// Example of "device-to-device" communication.
// [Notes]
// > Apply devices routes via "Diangnose / Device communication" in TerminalExplorer when PLC's are in run-mode.
//   Afterwards all communication errors will disappear. 
FUNCTION_BLOCK FB_Ref_PubSub_Remote EXTENDS FB_BA_View
VAR CONSTANT
	{region 'Test Settings'}
		// Use one (remote) device:
//		sDevice1_NetID			: T_BA_MedString				:= '192.168.10.100.1.1';
//		sDevice2_NetID			: T_BA_MedString				:= '192.168.10.100.1.1';
			 
		// Use one (loopback) device:
		sDevice1_NetID			: T_BA_MedString				:= '127.0.0.1.1.1';
		sDevice2_NetID			: T_BA_MedString				:= '127.0.0.1.1.1';
			 
		// Use two (remote and loopback) devices:
//		sDevice1_NetID			: T_BA_MedString				:= '192.168.2.200.1.1';
//		sDevice2_NetID			: T_BA_MedString				:= '127.0.0.1.1.1';
			 
		// Use two (remote) devices:
//		sDevice1_NetID			: T_BA_MedString				:= '192.168.10.100.1.1';
//		sDevice2_NetID			: T_BA_MedString				:= '192.168.2.200.1.1';
	{endregion}
END_VAR
VAR
	{region 'Analog'}
		AV_Sub					: FB_BA_SubAPrio := (
									sSubject					:= 'AV_Obj',
									sTarget						:= sDevice1_NetID,
									tReadInterval				:= T#5S								// Set shorter read interval
								);
		AVOp_Sub				: FB_BA_SubAV_Op := (
									sSubject					:= 'AVOp_Obj',
									sTarget						:= sDevice1_NetID,
									tReadInterval				:= T#5S								// Set shorter read interval
								);
		AI_Sub					: FB_BA_SubAI := (
									sSubject					:= 'AI_Obj',
									sTarget						:= sDevice2_NetID,
									tReadInterval				:= T#5S								// Set shorter read interval
								);
		AO_Sub					: FB_BA_SubAPrio := (
									sSubject					:= 'AO_Obj',
									sTarget						:= sDevice2_NetID,
									tReadInterval				:= T#5S								// Set shorter read interval
								);
	{endregion}
	{region 'Binary'}
		BV_Sub					: FB_BA_SubBPrio := (
									sSubject					:= 'BV_Obj',
									sTarget						:= sDevice1_NetID
								);
		BVOp_Sub				: FB_BA_SubBV_Op := (
									sSubject					:= 'BVOp_Obj',
									sTarget						:= sDevice1_NetID
								);
		BI_Sub					: FB_BA_SubBI := (
									sSubject					:= 'BI_Obj',
									sTarget						:= sDevice2_NetID
								);
		BO_Sub					: FB_BA_SubBPrio := (
									sSubject					:= 'BO_Obj',
									sTarget						:= sDevice2_NetID
								);
	{endregion}
	{region 'Multistate'}
		MV_Sub					: FB_BA_SubMPrio := (
									sSubject					:= 'MV_Obj',
									sTarget						:= sDevice1_NetID
								);
		MVOp_Sub				: FB_BA_SubMV_Op := (
									sSubject					:= 'MVOp_Obj',
									sTarget						:= sDevice1_NetID
								);
		MI_Sub					: FB_BA_SubMI := (
									sSubject					:= 'MI_Obj',
									sTarget						:= sDevice2_NetID
								);
		MO_Sub					: FB_BA_SubMPrio := (
									sSubject					:= 'MO_Obj',
									sTarget						:= sDevice2_NetID
								);
	{endregion}
	{region 'Multistate'}
		Loop_Sub				: FB_BA_SubLoop := (
									sSubject					:= 'Loop_Obj',
									sTarget						:= sDevice1_NetID
								);		
		Cal_Sub					: FB_BA_SubCal := (
									sSubject					:= 'Cal_Obj',
									sTarget						:= sDevice1_NetID
								);
		SchedA_Sub				: FB_BA_SubSchedA := (
									sSubject					:= 'SchedA_Obj',
									sTarget						:= sDevice1_NetID
								);
		SchedB_Sub				: FB_BA_SubSchedB := (
									sSubject					:= 'SchedB_Obj',
									sTarget						:= sDevice1_NetID
								);
		SchedM_Sub				: FB_BA_SubSchedM := (
									sSubject					:= 'SchedM_Obj',
									sTarget						:= sDevice1_NetID
								);
		Trend_Sub				: FB_BA_SubTrend := (
									sSubject					:= 'Trend_Obj',
									sTarget						:= sDevice2_NetID
								);
	{endregion}	  
	{region 'Custom'}
		{region 'Typed'}  
			MyWthSt1_Sub		: FB_BA_MyWeatherStationSub := (
									sSubject					:= 'MyWthSt',
									sTarget						:= sDevice1_NetID,
									tReadInterval				:= T#5S,							// Set shorter read interval
									tReadTolerance				:= T#20S,							// Tolerate read errors for a short time
									bClearOnReadError			:= TRUE								// Clear data on error
								);
			MyWthSt2_Sub		: FB_BA_MyWeatherStationSub := (
									sSubject					:= 'MyWthSt',
									sTarget						:= sDevice2_NetID
								);
			MyWthSt3_Sub		: FB_BA_MyWeatherStationSub := (
									sSubject					:= 'MyWthSt',
									sTarget						:= sDevice2_NetID
								);
		{endregion}
		{region 'Raw'}
			MyRawWthSt1Data_Sub	: ST_BA_MyWeatherData;
			MyRawWthSt1_Sub		: FB_BA_RawSubscriber := (
									sSubject					:= 'MyRawWthSt',
									sTarget						:= sDevice1_NetID
								);
			MyRawWthSt2Data_Sub	: ST_BA_MyWeatherData;
			MyRawWthSt2_Sub		: FB_BA_RawSubscriber := (
									sSubject					:= 'MyRawWthSt',
									sTarget						:= sDevice2_NetID
								);
		{endregion}
	{endregion} 
	{region 'Tests'}
		{region 'Subject path'}
			Nested1a_AV_Sub		: FB_BA_SubAV_Op := (
								//	sSubject					:= 'fbAV',							// -> Would lead to ambiguous subject!
									sSubject					:= 'Nested1a.Value',
									sTarget						:= sDevice1_NetID
								);
			Nested1b_AV_Sub		: FB_BA_SubAV_Op := (
								//	sSubject					:= 'fbAV',							// -> Would lead to ambiguous subject!
									sSubject					:= 'Nested1b.Value',
									sTarget						:= sDevice1_NetID
								);
		{endregion}
	{endregion}
END_VAR

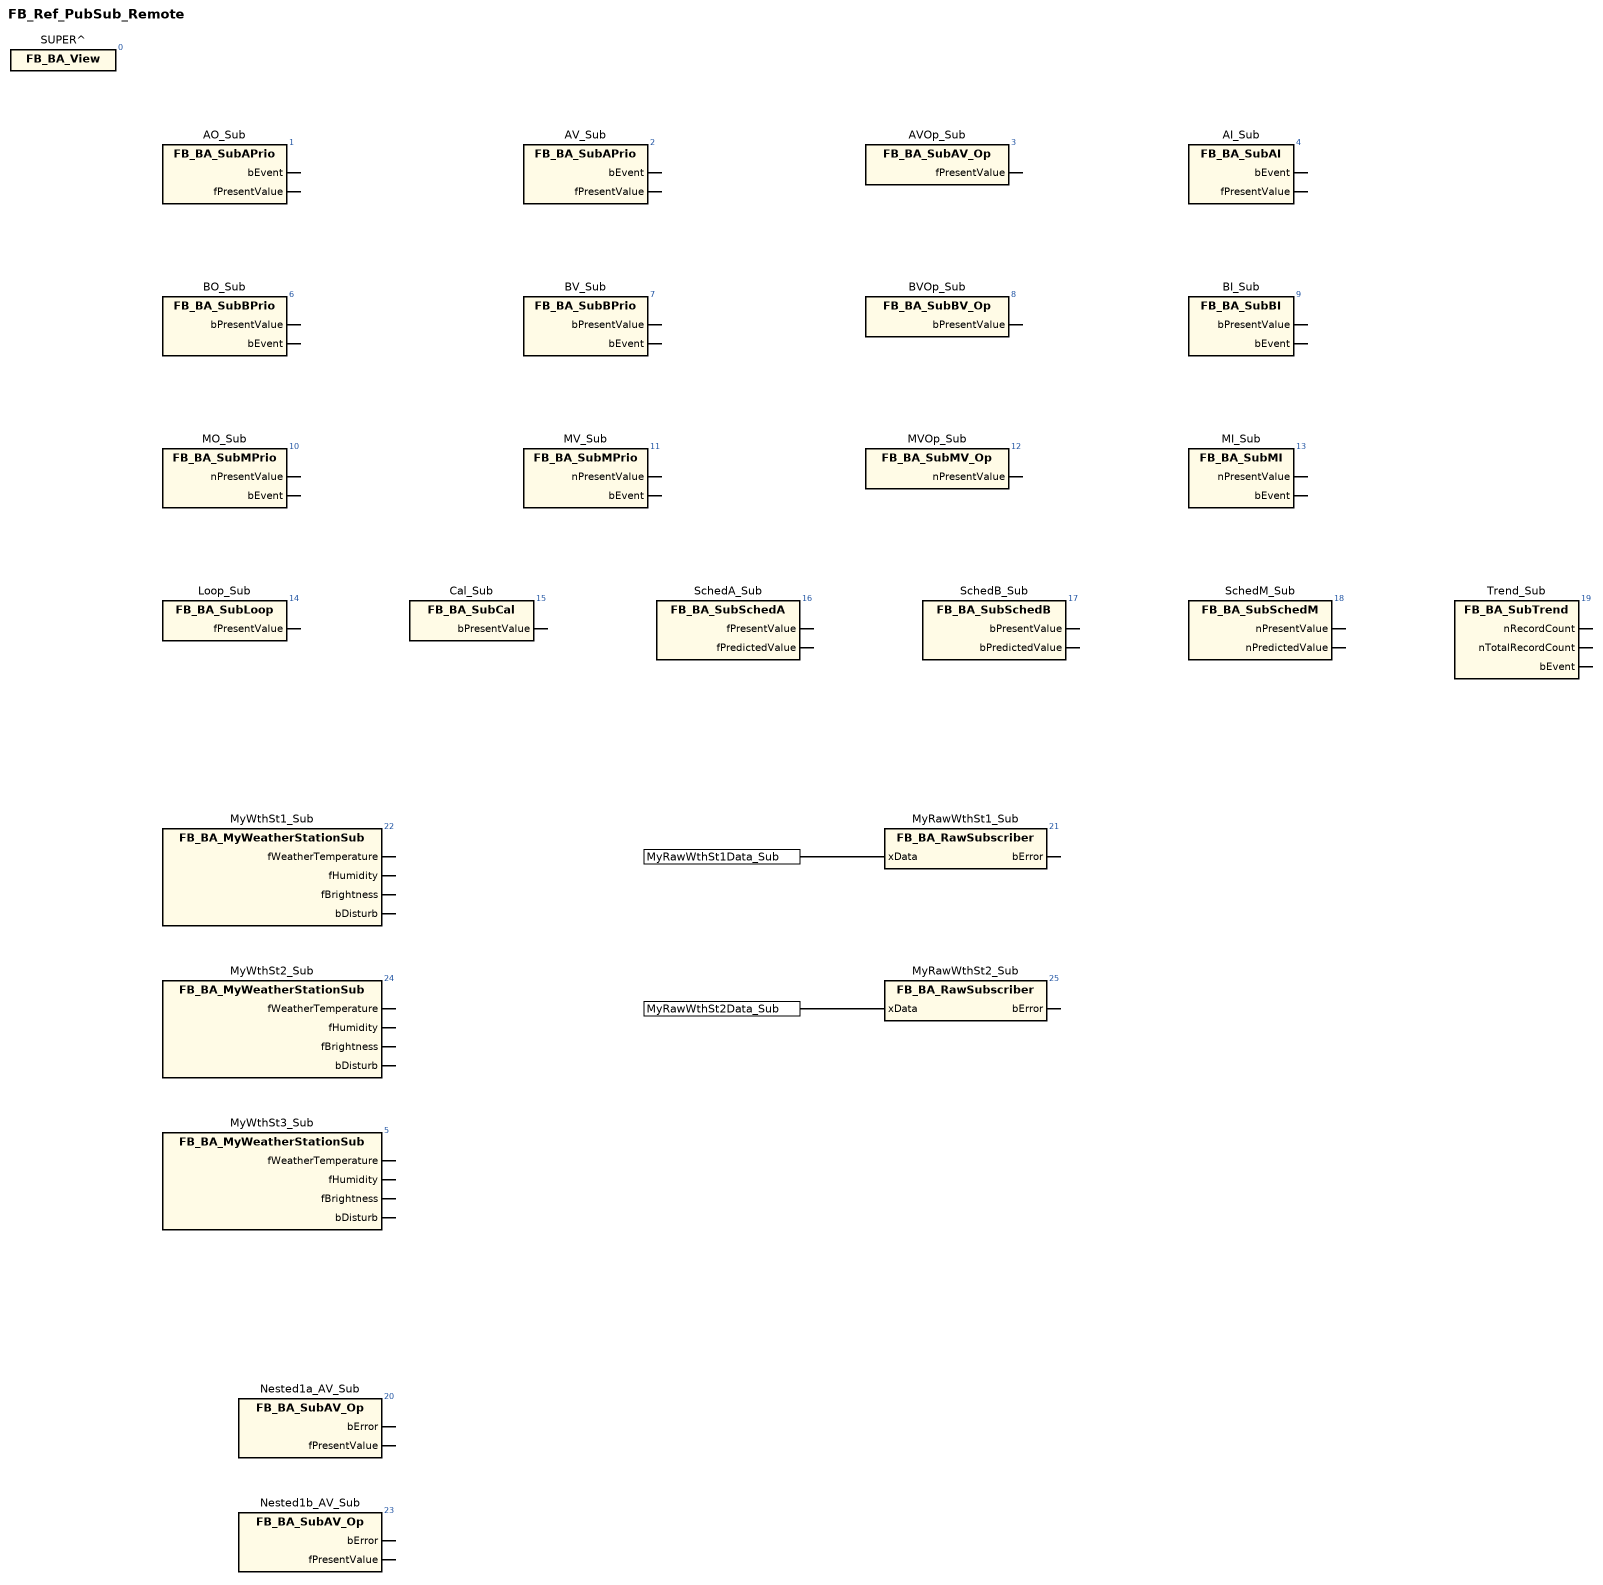
SUPER^(); // FB_BA_View
AO_Sub(); // FB_BA_SubAPrio
AV_Sub(); // FB_BA_SubAPrio
AVOp_Sub(); // FB_BA_SubAV_Op
AI_Sub(); // FB_BA_SubAI
MyWthSt3_Sub(); // FB_BA_MyWeatherStationSub
BO_Sub(); // FB_BA_SubBPrio
BV_Sub(); // FB_BA_SubBPrio
BVOp_Sub(); // FB_BA_SubBV_Op
BI_Sub(); // FB_BA_SubBI
MO_Sub(); // FB_BA_SubMPrio
MV_Sub(); // FB_BA_SubMPrio
MVOp_Sub(); // FB_BA_SubMV_Op
MI_Sub(); // FB_BA_SubMI
Loop_Sub(); // FB_BA_SubLoop
Cal_Sub(); // FB_BA_SubCal
SchedA_Sub(); // FB_BA_SubSchedA
SchedB_Sub(); // FB_BA_SubSchedB
SchedM_Sub(); // FB_BA_SubSchedM
Trend_Sub(); // FB_BA_SubTrend
Nested1a_AV_Sub(); // FB_BA_SubAV_Op
MyRawWthSt1_Sub(xData := MyRawWthSt1Data_Sub); // FB_BA_RawSubscriber
MyWthSt1_Sub(); // FB_BA_MyWeatherStationSub
Nested1b_AV_Sub(); // FB_BA_SubAV_Op
MyWthSt2_Sub(); // FB_BA_MyWeatherStationSub
MyRawWthSt2_Sub(xData := MyRawWthSt2Data_Sub); // FB_BA_RawSubscriber

END_FUNCTION_BLOCK

(* stored: Version 1.1.0.1, ProductVersion 3.1.4024.9
   POU FB_Ref_PubSub_Remote: Id {21c8c2c4-124a-41c0-a75b-a7da558bc577}, SpecialFunc None *)
